{attribute 'qualified_only'}
{attribute 'strict'}
TYPE StateSeparator :
(
	Off,
	Init,
	Init_Wait,
	Ready,
	Eject,
	Eject_Wait_1,
	Eject_Wait_2,
	Done_Wait,
	Done
);
END_TYPE

(* stored: Version 1.1.0.1, ProductVersion 3.1.4024.6
   DUT StateSeparator: Id {1267d366-f7fe-4571-a1b3-af3164a5ecbc} *)
